{attribute addProperty BoxType "EL2596-0000-0017"}
{attribute addProperty Id "ControlAT %Q*Control_4AC92B13162"}
{attribute addProperty CRC "857785697"}
{attribute addProperty SizeInBites "16"}
{attribute addProperty SizeInBytes "2"}
TYPE DOX_Control_3320C561 :
STRUCT
	{attribute addProperty Name "Control"}
	Control AT %Q* : Control_4AC92B13;
END_STRUCT
END_TYPE

(* stored: Version 1.2.0.0, ProductVersion 3.1.4024.9
   DUT DOX_Control_3320C561: Id {83f558fd-1678-47d9-b8b7-0dbd5393be72} *)
